Fanuc KAREL source: kt00564.KL

-- PROVISIONAL review KL for V1013-1; original PC SHA256 ab08f88fe304f1135dd566145e8b99662b19b581ae6473fe9184dffc460a54ac
-- Incomplete behavior may be omitted. Consult companion uncertainty JSON. Do not deploy.
PROGRAM KT00564
%NOLOCKGROUP
VAR
  OUT : REAL
-- UNRESOLVED_DECL V1 type=000013
-- UNRESOLVED_DECL V2 type=000013
BEGIN
  -- UNRESOLVED_PC offsets 5-20; opcodes 2E,22,32,35
  -- UNRESOLVED_PC offsets 25-40; opcodes 2E,22,32,35
  -- UNRESOLVED_PC offsets 45-60; opcodes 2E,22,32,35
  -- UNRESOLVED_PC offsets 65-80; opcodes 2E,22,32,35
  -- UNRESOLVED_PC offsets 85-108; opcodes 49,49,94,23
  -- UNRESOLVED_PC offsets 113-117; opcodes 7F
END KT00564
